// TIA Portal V18 export
FUNCTION "Datalog" : Void   // FC13, LAD
{ S7_Optimized_Access := 'TRUE' }
VERSION : 0.1
// stored: AutoNumber true, IsIECCheckEnabled false, SetENOAutomatically false, UDAEnableTagReadback false
   VAR_TEMP
      "return" : Int;
   END_VAR
   VAR_TEMP   // added for the SCL form of the ladder/FBD networks
      _w1 : Bool;
      _w2 : Bool;
      _w3 : Bool;
      _w4 : Bool;
      _w5 : Bool;
      _w6 : Bool;
      _w7 : Bool;
      _w8 : Bool;
   END_VAR
BEGIN

REGION Network 1
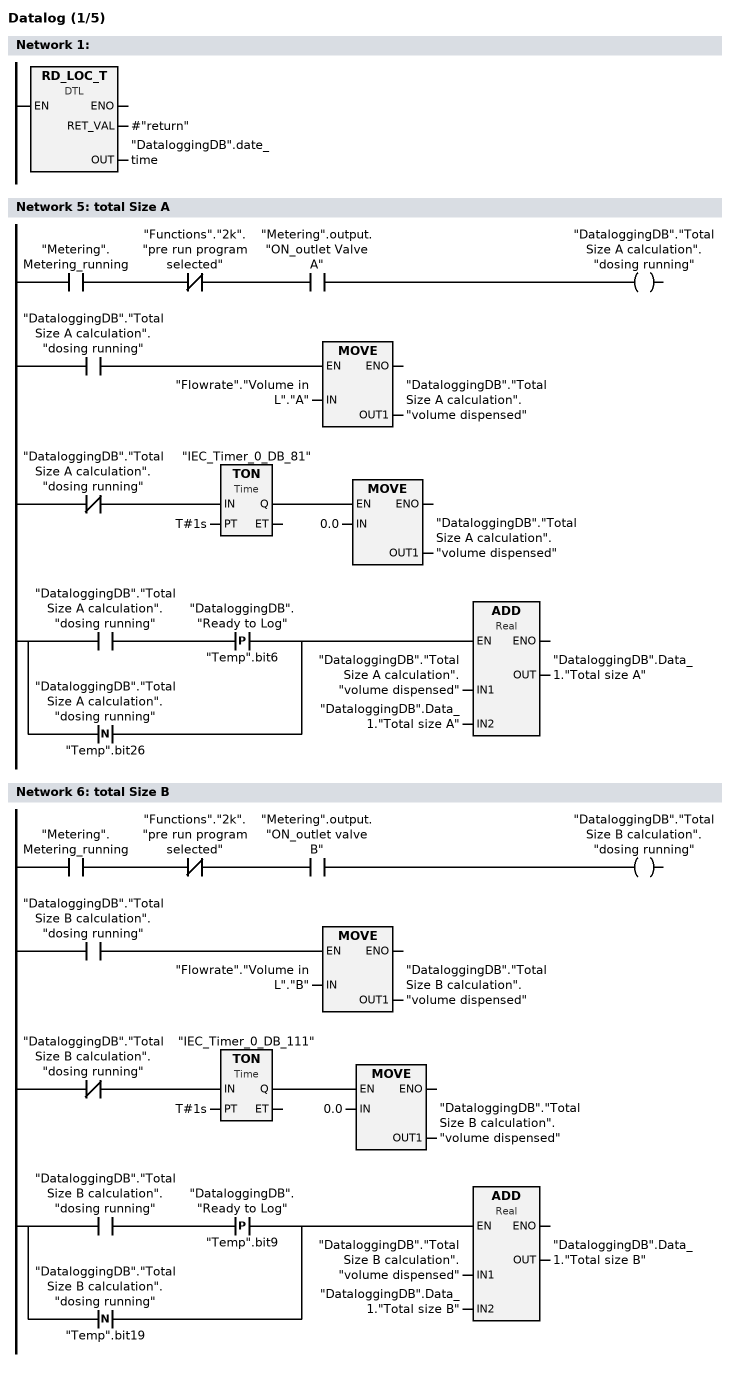
   RUNG wire#powerrail
      { S7_Templates := "date_type := DTL" } RD_LOC_T(RET_VAL => #"return", OUT => "DataloggingDB".date_time)
   END_RUNG
   // the same network as SCL:
   #"return" := RD_LOC_T(OUT => "DataloggingDB".date_time);
END_REGION

REGION Network 2 (SCL)
   IF "DataloggingDB".date_time.DAY <> "DataloggingDB".previous_day THEN
       //"DataloggingDB".day_changed := true;
       "DataloggingDB".totalsizepreviousday:="DataloggingDB".Data_1."Total Size";
       "DataloggingDB".previous_day := "DataloggingDB".date_time.DAY ;
   ELSE
       "DataloggingDB".day_changed := false;
   END_IF;
   IF "DataloggingDB".current_week <> "DataloggingDB".previous_week THEN
       //"DataloggingDB".day_changed := true;
       "DataloggingDB".totalsizepreviousweek := "DataloggingDB".Data_1."Total Size";
       "DataloggingDB".previous_week := "DataloggingDB".current_week;
   ELSE
       "DataloggingDB".day_changed := false;
   END_IF;

   IF "DataloggingDB".date_time.MONTH <> "DataloggingDB".previous_month THEN
       //"DataloggingDB".month_changed := true;
       "DataloggingDB".totalsizepreviousmonth := "DataloggingDB".Data_1."Total Size";
       "DataloggingDB".previous_month := "DataloggingDB".date_time.MONTH;
   ELSE
       "DataloggingDB".month_changed := false;
   END_IF;

   "DataloggingDB".totalsizeday := "DataloggingDB".Data_1."Total Size" - "DataloggingDB".totalsizepreviousday ;
   "DataloggingDB".totalsizeweek := "DataloggingDB".Data_1."Total Size" - "DataloggingDB".totalsizepreviousweek;
   "DataloggingDB".totalsizemonth := "DataloggingDB".Data_1."Total Size" - "DataloggingDB".totalsizepreviousmonth;
END_REGION

REGION Network 3 (SCL): Total Flush A
   IF (("Function Flush"."Control A"."flush running" AND "Functions"."flush selection"."Flush A selected") OR
       "Function Regenaration PGM".Control."metering running" OR
       "Function Ratio check".Control."metering running" OR
       ("Functions"."2k"."pre run program selected" AND "Metering".Metering_running) OR
       "Function Dearing with valve"."Control A"."dearing running") THEN
       "DataloggingDB"."Copy Flush A qty" := true;
   END_IF;

   "R_TRIG_DB_1"(CLK:="DataloggingDB"."Copy Flush A qty" AND NOT ("Function Dearing with valve"."Control A"."dearing running") AND
                 NOT ("Function Regenaration PGM".Control."metering running") AND NOT ("Function Ratio check".Control."metering running") AND
                 NOT ("Functions"."2k"."pre run program selected") AND NOT ("Function Flush"."Control A"."flush running"),
                 Q=>"Temp".bit1);

   IF "R_TRIG_DB_1".Q THEN
       "DataloggingDB".Data_1."Total A flush" := "Flowrate"."Volume in L".mixed +"DataloggingDB".Data_1."Total A flush";
       "DataloggingDB"."Copy Flush A qty" := false;
   END_IF;
END_REGION

REGION Network 4 (SCL)
   IF (("Function Flush"."Control B"."flush running" AND "Functions"."flush selection"."Flush B selected") OR
       "Function Regenaration PGM".Control."metering running" OR
       "Function Ratio check".Control."metering running" OR
       ("Functions"."2k"."pre run program selected" AND "Metering".Metering_running) OR
       "Function Dearing with valve"."Control B"."dearing running") THEN
       "DataloggingDB"."Copy Flush B qty" := true;
   END_IF;

   "R_TRIG_DB_21"(CLK:="DataloggingDB"."Copy Flush B qty" AND NOT ("Function Dearing with valve"."Control B"."dearing running") AND
                  NOT ("Function Regenaration PGM".Control."metering running") AND NOT ("Function Ratio check".Control."metering running") AND
                  NOT ("Functions"."2k"."pre run program selected") AND NOT ("Function Flush"."Control B"."flush running"),
                  Q=>"Temp".bit3);

   IF "R_TRIG_DB_21".Q THEN
       "DataloggingDB".Data_1."Total B flush" := "Flowrate"."Volume in L".mixed + "DataloggingDB".Data_1."Total B flush";
       "DataloggingDB"."Copy Flush B qty" := false;
   END_IF;
END_REGION

REGION Network 5: total Size A
   RUNG wire#powerrail
      Contact( "Metering".Metering_running )
      I_Contact( "Functions"."2k"."pre run program selected" )
      Contact( "Metering".output."ON_outlet Valve A" )
      Coil( "DataloggingDB"."Total Size A calculation"."dosing running" )
   END_RUNG
   RUNG wire#powerrail
      Contact( "DataloggingDB"."Total Size A calculation"."dosing running" )
      Move(in := "Flowrate"."Volume in L"."A", out1 => "DataloggingDB"."Total Size A calculation"."volume dispensed")
   END_RUNG
   RUNG wire#powerrail
      I_Contact( "DataloggingDB"."Total Size A calculation"."dosing running" )
      { S7_Templates := "time_type := Time" } "IEC_Timer_0_DB_81".TON(pt := T#1s, et =>)
      Move(in := 0.0, out1 => "DataloggingDB"."Total Size A calculation"."volume dispensed")
   END_RUNG
   RUNG wire#powerrail
      Contact( "DataloggingDB"."Total Size A calculation"."dosing running" )
      P_Contact(operand := "DataloggingDB"."Ready to Log", bit := "Temp".bit6)
      wire#w1
      { S7_Templates := "SrcType := Real" } Add(in1 := "DataloggingDB"."Total Size A calculation"."volume dispensed", in2 := "DataloggingDB".Data_1."Total size A", out => "DataloggingDB".Data_1."Total size A")
   END_RUNG
   RUNG wire#powerrail
      N_Contact(operand := "DataloggingDB"."Total Size A calculation"."dosing running", bit := "Temp".bit26)
   END_RUNG wire#w1
   // the same network as SCL:
   "DataloggingDB"."Total Size A calculation"."dosing running" := "Metering".Metering_running AND NOT "Functions"."2k"."pre run program selected" AND "Metering".output."ON_outlet Valve A";
   IF "DataloggingDB"."Total Size A calculation"."dosing running" THEN
       "DataloggingDB"."Total Size A calculation"."volume dispensed" := "Flowrate"."Volume in L"."A";
   END_IF;
   "IEC_Timer_0_DB_81".TON(IN := NOT "DataloggingDB"."Total Size A calculation"."dosing running", PT := T#1s);
   IF "IEC_Timer_0_DB_81".Q THEN
       "DataloggingDB"."Total Size A calculation"."volume dispensed" := 0.0;
   END_IF;
   #_w1 := "DataloggingDB"."Total Size A calculation"."dosing running" AND "DataloggingDB"."Ready to Log" AND NOT "Temp".bit6;   // rising edge of "DataloggingDB"."Ready to Log"
   "Temp".bit6 := "DataloggingDB"."Ready to Log";
   #_w2 := NOT "DataloggingDB"."Total Size A calculation"."dosing running" AND "Temp".bit26;   // falling edge of "DataloggingDB"."Total Size A calculation"."dosing running"
   "Temp".bit26 := "DataloggingDB"."Total Size A calculation"."dosing running";
   IF #_w1 OR #_w2 THEN
       "DataloggingDB".Data_1."Total size A" := "DataloggingDB"."Total Size A calculation"."volume dispensed" + "DataloggingDB".Data_1."Total size A";
   END_IF;
END_REGION

REGION Network 6: total Size B
   RUNG wire#powerrail
      Contact( "Metering".Metering_running )
      I_Contact( "Functions"."2k"."pre run program selected" )
      Contact( "Metering".output."ON_outlet valve B" )
      Coil( "DataloggingDB"."Total Size B calculation"."dosing running" )
   END_RUNG
   RUNG wire#powerrail
      Contact( "DataloggingDB"."Total Size B calculation"."dosing running" )
      Move(in := "Flowrate"."Volume in L"."B", out1 => "DataloggingDB"."Total Size B calculation"."volume dispensed")
   END_RUNG
   RUNG wire#powerrail
      I_Contact( "DataloggingDB"."Total Size B calculation"."dosing running" )
      { S7_Templates := "time_type := Time" } "IEC_Timer_0_DB_111".TON(pt := T#1s, et =>)
      Move(in := 0.0, out1 => "DataloggingDB"."Total Size B calculation"."volume dispensed")
   END_RUNG
   RUNG wire#powerrail
      Contact( "DataloggingDB"."Total Size B calculation"."dosing running" )
      P_Contact(operand := "DataloggingDB"."Ready to Log", bit := "Temp".bit9)
      wire#w1
      { S7_Templates := "SrcType := Real" } Add(in1 := "DataloggingDB"."Total Size B calculation"."volume dispensed", in2 := "DataloggingDB".Data_1."Total size B", out => "DataloggingDB".Data_1."Total size B")
   END_RUNG
   RUNG wire#powerrail
      N_Contact(operand := "DataloggingDB"."Total Size B calculation"."dosing running", bit := "Temp".bit19)
   END_RUNG wire#w1
   // the same network as SCL:
   "DataloggingDB"."Total Size B calculation"."dosing running" := "Metering".Metering_running AND NOT "Functions"."2k"."pre run program selected" AND "Metering".output."ON_outlet valve B";
   IF "DataloggingDB"."Total Size B calculation"."dosing running" THEN
       "DataloggingDB"."Total Size B calculation"."volume dispensed" := "Flowrate"."Volume in L"."B";
   END_IF;
   "IEC_Timer_0_DB_111".TON(IN := NOT "DataloggingDB"."Total Size B calculation"."dosing running", PT := T#1s);
   IF "IEC_Timer_0_DB_111".Q THEN
       "DataloggingDB"."Total Size B calculation"."volume dispensed" := 0.0;
   END_IF;
   #_w1 := "DataloggingDB"."Total Size B calculation"."dosing running" AND "DataloggingDB"."Ready to Log" AND NOT "Temp".bit9;   // rising edge of "DataloggingDB"."Ready to Log"
   "Temp".bit9 := "DataloggingDB"."Ready to Log";
   #_w2 := NOT "DataloggingDB"."Total Size B calculation"."dosing running" AND "Temp".bit19;   // falling edge of "DataloggingDB"."Total Size B calculation"."dosing running"
   "Temp".bit19 := "DataloggingDB"."Total Size B calculation"."dosing running";
   IF #_w1 OR #_w2 THEN
       "DataloggingDB".Data_1."Total size B" := "DataloggingDB"."Total Size B calculation"."volume dispensed" + "DataloggingDB".Data_1."Total size B";
   END_IF;
END_REGION

REGION Network 7: Total size
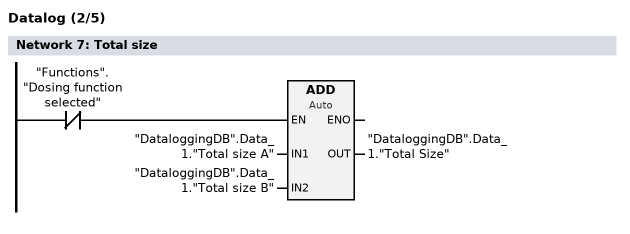
   RUNG wire#powerrail
      I_Contact( "Functions"."Dosing function selected" )
      Add(in1 := "DataloggingDB".Data_1."Total size A", in2 := "DataloggingDB".Data_1."Total size B", out => "DataloggingDB".Data_1."Total Size")
   END_RUNG
   // the same network as SCL:
   IF NOT "Functions"."Dosing function selected" THEN
       "DataloggingDB".Data_1."Total Size" := "DataloggingDB".Data_1."Total size A" + "DataloggingDB".Data_1."Total size B";
   END_IF;
END_REGION

REGION Network 8: Metering Size
END_REGION

REGION Network 9: Shot Size A
END_REGION

REGION Network 10: Shot Size B
END_REGION

REGION Network 11: Mixing Ratio
END_REGION

REGION Network 12: ratio Min
END_REGION

REGION Network 13: ratio Max
END_REGION

REGION Network 14: Volume_Dispensed
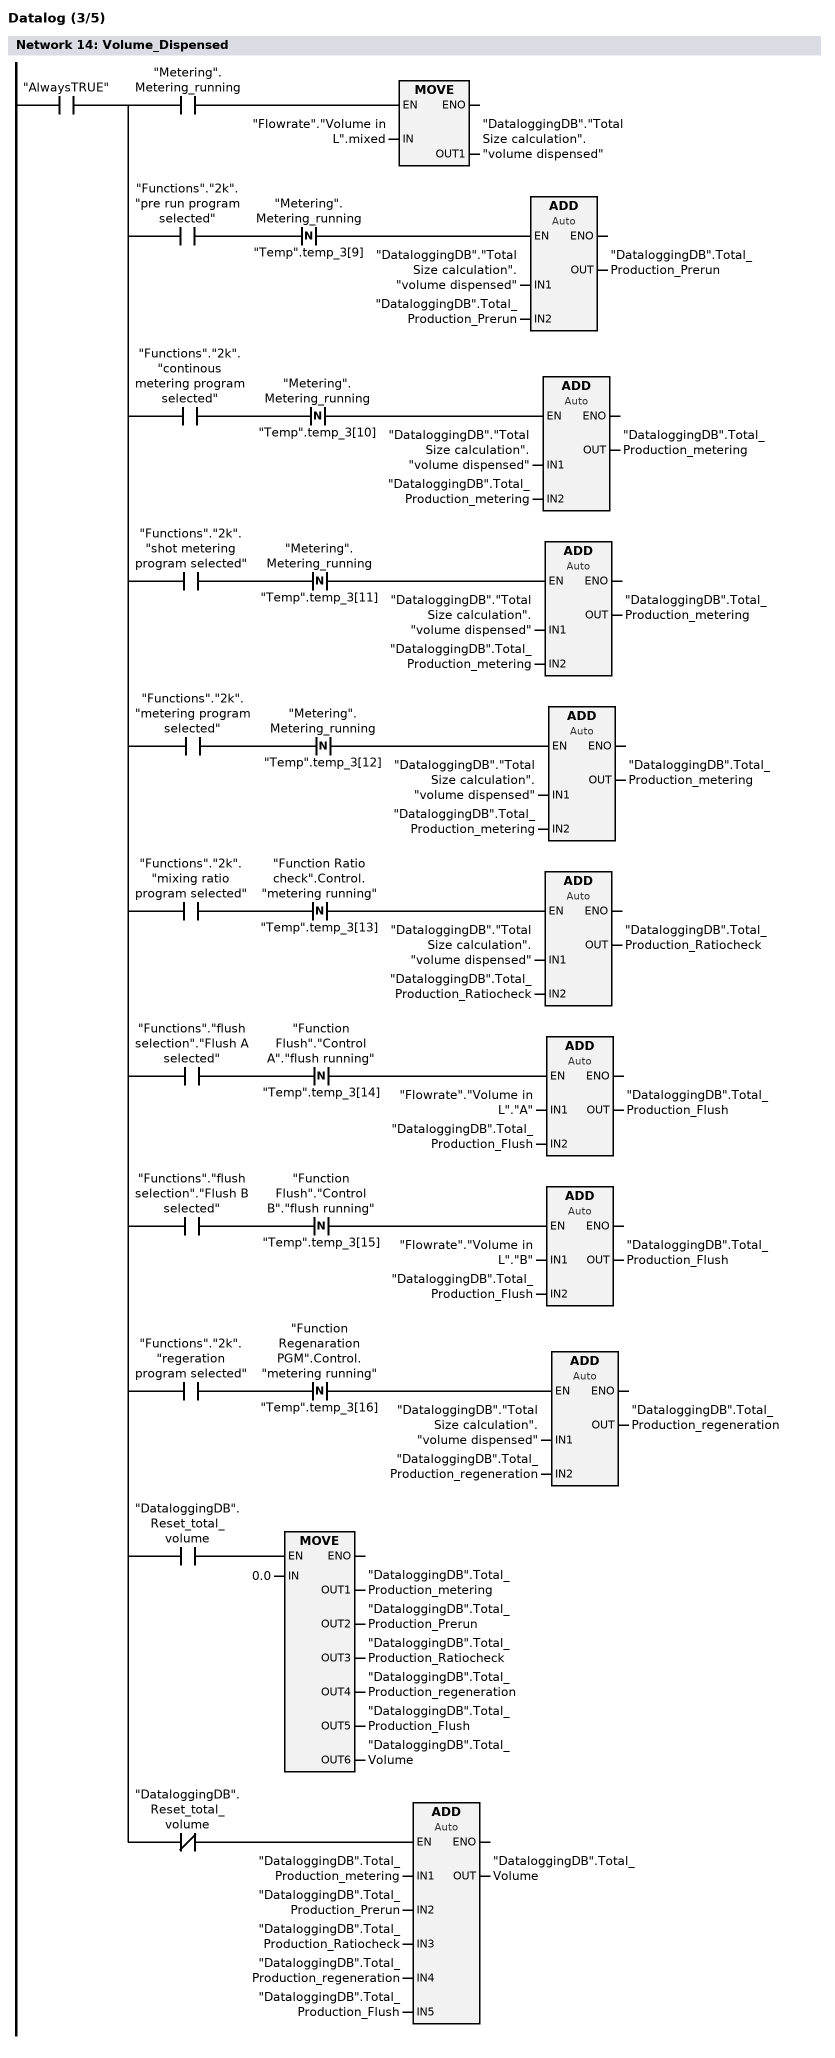
   RUNG wire#powerrail
      Contact( "AlwaysTRUE" )
      wire#w1
      Contact( "Metering".Metering_running )
      Move(in := "Flowrate"."Volume in L".mixed, out1 => "DataloggingDB"."Total Size calculation"."volume dispensed")
   END_RUNG
   RUNG wire#w1
      Contact( "Functions"."2k"."pre run program selected" )
      N_Contact(operand := "Metering".Metering_running, bit := "Temp".temp_3[9])
      Add(in1 := "DataloggingDB"."Total Size calculation"."volume dispensed", in2 := "DataloggingDB".Total_Production_Prerun, out => "DataloggingDB".Total_Production_Prerun)
   END_RUNG
   RUNG wire#w1
      Contact( "Functions"."2k"."continous metering program selected" )
      N_Contact(operand := "Metering".Metering_running, bit := "Temp".temp_3[10])
      Add(in1 := "DataloggingDB"."Total Size calculation"."volume dispensed", in2 := "DataloggingDB".Total_Production_metering, out => "DataloggingDB".Total_Production_metering)
   END_RUNG
   RUNG wire#w1
      Contact( "Functions"."2k"."shot metering program selected" )
      N_Contact(operand := "Metering".Metering_running, bit := "Temp".temp_3[11])
      Add(in1 := "DataloggingDB"."Total Size calculation"."volume dispensed", in2 := "DataloggingDB".Total_Production_metering, out => "DataloggingDB".Total_Production_metering)
   END_RUNG
   RUNG wire#w1
      Contact( "Functions"."2k"."metering program selected" )
      N_Contact(operand := "Metering".Metering_running, bit := "Temp".temp_3[12])
      Add(in1 := "DataloggingDB"."Total Size calculation"."volume dispensed", in2 := "DataloggingDB".Total_Production_metering, out => "DataloggingDB".Total_Production_metering)
   END_RUNG
   RUNG wire#w1
      Contact( "Functions"."2k"."mixing ratio program selected" )
      N_Contact(operand := "Function Ratio check".Control."metering running", bit := "Temp".temp_3[13])
      Add(in1 := "DataloggingDB"."Total Size calculation"."volume dispensed", in2 := "DataloggingDB".Total_Production_Ratiocheck, out => "DataloggingDB".Total_Production_Ratiocheck)
   END_RUNG
   RUNG wire#w1
      Contact( "Functions"."flush selection"."Flush A selected" )
      N_Contact(operand := "Function Flush"."Control A"."flush running", bit := "Temp".temp_3[14])
      Add(in1 := "Flowrate"."Volume in L"."A", in2 := "DataloggingDB".Total_Production_Flush, out => "DataloggingDB".Total_Production_Flush)
   END_RUNG
   RUNG wire#w1
      Contact( "Functions"."flush selection"."Flush B selected" )
      N_Contact(operand := "Function Flush"."Control B"."flush running", bit := "Temp".temp_3[15])
      Add(in1 := "Flowrate"."Volume in L"."B", in2 := "DataloggingDB".Total_Production_Flush, out => "DataloggingDB".Total_Production_Flush)
   END_RUNG
   RUNG wire#w1
      Contact( "Functions"."2k"."regeration program selected" )
      N_Contact(operand := "Function Regenaration PGM".Control."metering running", bit := "Temp".temp_3[16])
      Add(in1 := "DataloggingDB"."Total Size calculation"."volume dispensed", in2 := "DataloggingDB".Total_Production_regeneration, out => "DataloggingDB".Total_Production_regeneration)
   END_RUNG
   RUNG wire#w1
      Contact( "DataloggingDB".Reset_total_volume )
      Move(in := 0.0, out1 => "DataloggingDB".Total_Production_metering, out2 => "DataloggingDB".Total_Production_Prerun, out3 => "DataloggingDB".Total_Production_Ratiocheck, out4 => "DataloggingDB".Total_Production_regeneration, out5 => "DataloggingDB".Total_Production_Flush, out6 => "DataloggingDB".Total_Volume)
   END_RUNG
   RUNG wire#w1
      I_Contact( "DataloggingDB".Reset_total_volume )
      Add(in1 := "DataloggingDB".Total_Production_metering, in2 := "DataloggingDB".Total_Production_Prerun, in3 := "DataloggingDB".Total_Production_Ratiocheck, in4 := "DataloggingDB".Total_Production_regeneration, in5 := "DataloggingDB".Total_Production_Flush, out => "DataloggingDB".Total_Volume)
   END_RUNG
   // the same network as SCL:
   IF "AlwaysTRUE" AND "Metering".Metering_running THEN
       "DataloggingDB"."Total Size calculation"."volume dispensed" := "Flowrate"."Volume in L".mixed;
   END_IF;
   #_w1 := "AlwaysTRUE" AND "Functions"."2k"."pre run program selected" AND NOT "Metering".Metering_running AND "Temp".temp_3[9];   // falling edge of "Metering".Metering_running
   "Temp".temp_3[9] := "Metering".Metering_running;
   IF #_w1 THEN
       "DataloggingDB".Total_Production_Prerun := "DataloggingDB"."Total Size calculation"."volume dispensed" + "DataloggingDB".Total_Production_Prerun;
   END_IF;
   #_w2 := "AlwaysTRUE" AND "Functions"."2k"."continous metering program selected" AND NOT "Metering".Metering_running AND "Temp".temp_3[10];   // falling edge of "Metering".Metering_running
   "Temp".temp_3[10] := "Metering".Metering_running;
   IF #_w2 THEN
       "DataloggingDB".Total_Production_metering := "DataloggingDB"."Total Size calculation"."volume dispensed" + "DataloggingDB".Total_Production_metering;
   END_IF;
   #_w3 := "AlwaysTRUE" AND "Functions"."2k"."shot metering program selected" AND NOT "Metering".Metering_running AND "Temp".temp_3[11];   // falling edge of "Metering".Metering_running
   "Temp".temp_3[11] := "Metering".Metering_running;
   IF #_w3 THEN
       "DataloggingDB".Total_Production_metering := "DataloggingDB"."Total Size calculation"."volume dispensed" + "DataloggingDB".Total_Production_metering;
   END_IF;
   #_w4 := "AlwaysTRUE" AND "Functions"."2k"."metering program selected" AND NOT "Metering".Metering_running AND "Temp".temp_3[12];   // falling edge of "Metering".Metering_running
   "Temp".temp_3[12] := "Metering".Metering_running;
   IF #_w4 THEN
       "DataloggingDB".Total_Production_metering := "DataloggingDB"."Total Size calculation"."volume dispensed" + "DataloggingDB".Total_Production_metering;
   END_IF;
   #_w5 := "AlwaysTRUE" AND "Functions"."2k"."mixing ratio program selected" AND NOT "Function Ratio check".Control."metering running" AND "Temp".temp_3[13];   // falling edge of "Function Ratio check".Control."metering running"
   "Temp".temp_3[13] := "Function Ratio check".Control."metering running";
   IF #_w5 THEN
       "DataloggingDB".Total_Production_Ratiocheck := "DataloggingDB"."Total Size calculation"."volume dispensed" + "DataloggingDB".Total_Production_Ratiocheck;
   END_IF;
   #_w6 := "AlwaysTRUE" AND "Functions"."flush selection"."Flush A selected" AND NOT "Function Flush"."Control A"."flush running" AND "Temp".temp_3[14];   // falling edge of "Function Flush"."Control A"."flush running"
   "Temp".temp_3[14] := "Function Flush"."Control A"."flush running";
   IF #_w6 THEN
       "DataloggingDB".Total_Production_Flush := "Flowrate"."Volume in L"."A" + "DataloggingDB".Total_Production_Flush;
   END_IF;
   #_w7 := "AlwaysTRUE" AND "Functions"."flush selection"."Flush B selected" AND NOT "Function Flush"."Control B"."flush running" AND "Temp".temp_3[15];   // falling edge of "Function Flush"."Control B"."flush running"
   "Temp".temp_3[15] := "Function Flush"."Control B"."flush running";
   IF #_w7 THEN
       "DataloggingDB".Total_Production_Flush := "Flowrate"."Volume in L"."B" + "DataloggingDB".Total_Production_Flush;
   END_IF;
   #_w8 := "AlwaysTRUE" AND "Functions"."2k"."regeration program selected" AND NOT "Function Regenaration PGM".Control."metering running" AND "Temp".temp_3[16];   // falling edge of "Function Regenaration PGM".Control."metering running"
   "Temp".temp_3[16] := "Function Regenaration PGM".Control."metering running";
   IF #_w8 THEN
       "DataloggingDB".Total_Production_regeneration := "DataloggingDB"."Total Size calculation"."volume dispensed" + "DataloggingDB".Total_Production_regeneration;
   END_IF;
   IF "AlwaysTRUE" AND "DataloggingDB".Reset_total_volume THEN
       "DataloggingDB".Total_Production_metering := 0.0;
       "DataloggingDB".Total_Production_Prerun := 0.0;
       "DataloggingDB".Total_Production_Ratiocheck := 0.0;
       "DataloggingDB".Total_Production_regeneration := 0.0;
       "DataloggingDB".Total_Production_Flush := 0.0;
       "DataloggingDB".Total_Volume := 0.0;
   END_IF;
   IF "AlwaysTRUE" AND NOT "DataloggingDB".Reset_total_volume THEN
       "DataloggingDB".Total_Volume := "DataloggingDB".Total_Production_metering + "DataloggingDB".Total_Production_Prerun + "DataloggingDB".Total_Production_Ratiocheck + "DataloggingDB".Total_Production_regeneration + "DataloggingDB".Total_Production_Flush;
   END_IF;
END_REGION

REGION Network 15 (SCL)
   IF NOT ("Functions"."Dosing Running") THEN
       "event For datalogging"."event number" := 1; //Event machine idle
   ELSIF "Functions"."2k"."metering program selected" AND "Metering".Metering_running THEN
       "event For datalogging"."event number" := 2; //Event metering program running
   ELSIF "Function Ratio check".Control."metering running" THEN
       "event For datalogging"."event number" := 3; //Event Ratio check program running
   ELSIF "Functions"."2k"."shot metering program selected" AND "Metering".Metering_running THEN
       "event For datalogging"."event number" := 4; //Event metering shot running
   ELSIF "Functions"."2k"."continous metering program selected" AND "Metering".Metering_running THEN
       "event For datalogging"."event number" := 5; //Event metering Continuous metering running
   ELSIF "Functions"."2k"."pre run program selected" AND "Metering".Metering_running THEN
       "event For datalogging"."event number" := 6; //Event "Metering" Pre run running
   ELSIF "Function Flush"."Control A"."flush running" THEN
       "event For datalogging"."event number" := 7; // Event metering Flush running
   ELSIF "Function Dearing with valve"."Control A"."dearing running" OR "Function Dearing with valve"."Control B"."dearing running" THEN
       "event For datalogging"."event number" := 8; // Event deaerate running
   ELSIF "Faults&warnings"."Critical Alarm metering A&B" THEN
       "event For datalogging"."event number" := 9; // Event Machine fault
   ELSIF "Function Regenaration PGM".Control."metering running" THEN
       "event For datalogging"."event number" := 11; // Event regeneration running
   ELSIF "metering Completed" THEN
       "event For datalogging"."event number" := 12; // dosing completed
   END_IF;

   "DataloggingDB".Data.Function := "event For datalogging".Function_String["event For datalogging"."event number"];
END_REGION

REGION Network 16: Function
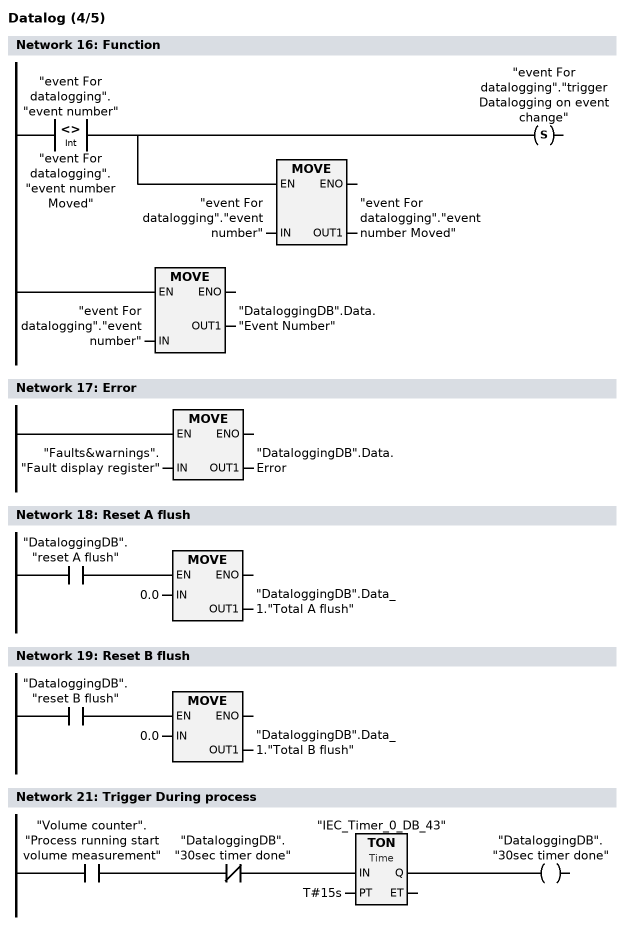
   RUNG wire#powerrail
      { S7_Templates := "SrcType := Int" } NE_Contact(in1 := "event For datalogging"."event number", in2 := "event For datalogging"."event number Moved")
      wire#w1
      S_Coil( "event For datalogging"."trigger Datalogging on event change" )
   END_RUNG
   RUNG wire#w1
      Move(in := "event For datalogging"."event number", out1 => "event For datalogging"."event number Moved")
   END_RUNG
   RUNG wire#powerrail
      Move(in := "event For datalogging"."event number", out1 => "DataloggingDB".Data."Event Number")
   END_RUNG
   // the same network as SCL:
   IF "event For datalogging"."event number" <> "event For datalogging"."event number Moved" THEN
       "event For datalogging"."trigger Datalogging on event change" := TRUE;
       "event For datalogging"."event number Moved" := "event For datalogging"."event number";
   END_IF;
   "DataloggingDB".Data."Event Number" := "event For datalogging"."event number";
END_REGION

REGION Network 17: Error
   RUNG wire#powerrail
      Move(in := "Faults&warnings"."Fault display register", out1 => "DataloggingDB".Data.Error)
   END_RUNG
   // the same network as SCL:
   "DataloggingDB".Data.Error := "Faults&warnings"."Fault display register";
END_REGION

REGION Network 18: Reset A flush
   RUNG wire#powerrail
      Contact( "DataloggingDB"."reset A flush" )
      Move(in := 0.0, out1 => "DataloggingDB".Data_1."Total A flush")
   END_RUNG
   // the same network as SCL:
   IF "DataloggingDB"."reset A flush" THEN "DataloggingDB".Data_1."Total A flush" := 0.0; END_IF;
END_REGION

REGION Network 19: Reset B flush
   RUNG wire#powerrail
      Contact( "DataloggingDB"."reset B flush" )
      Move(in := 0.0, out1 => "DataloggingDB".Data_1."Total B flush")
   END_RUNG
   // the same network as SCL:
   IF "DataloggingDB"."reset B flush" THEN "DataloggingDB".Data_1."Total B flush" := 0.0; END_IF;
END_REGION

REGION Network 20 (SCL): Reset total size
   IF "DataloggingDB"."reset total Size" THEN
       "DataloggingDB".Data_1."Total size A" := 0;
       "DataloggingDB".Data_1."Total size B" := 0;
       "DataloggingDB".totalsizeday := 0;
       "DataloggingDB".totalsizepreviousday := 0;
       "DataloggingDB".totalsizeweek := 0;
       "DataloggingDB".totalsizepreviousweek := 0;
       "DataloggingDB".totalsizemonth := 0;
       "DataloggingDB".totalsizepreviousmonth := 0;
       "DataloggingDB"."reset total Size" := FALSE;
   END_IF;
END_REGION

REGION Network 21: Trigger During process
   RUNG wire#powerrail
      Contact( "Volume counter"."Process running start volume measurement" )
      I_Contact( "DataloggingDB"."30sec timer done" )
      { S7_Templates := "time_type := Time" } "IEC_Timer_0_DB_43".TON(pt := T#15s, et =>)
      Coil( "DataloggingDB"."30sec timer done" )
   END_RUNG
   // the same network as SCL:
   "IEC_Timer_0_DB_43".TON(IN := "Volume counter"."Process running start volume measurement" AND NOT "DataloggingDB"."30sec timer done",
                           PT := T#15s);
   "DataloggingDB"."30sec timer done" := "IEC_Timer_0_DB_43".Q;
END_REGION

REGION Network 22: trigger data logging
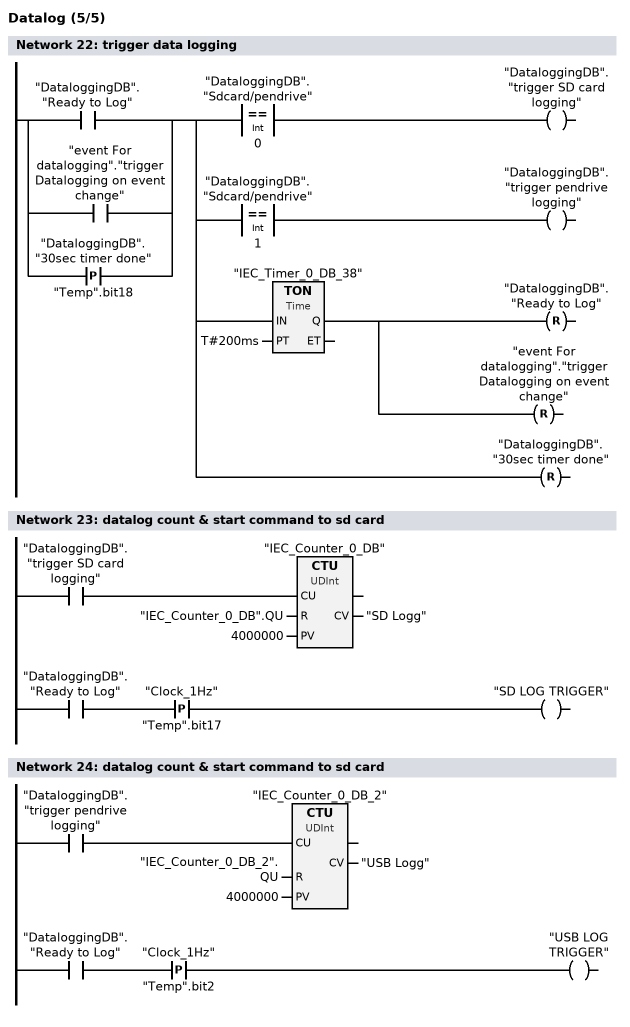
   RUNG wire#powerrail
      Contact( "DataloggingDB"."Ready to Log" )
      wire#w1
      { S7_Templates := "SrcType := Int" } EQ_Contact(in1 := "DataloggingDB"."Sdcard/pendrive", in2 := 0)
      Coil( "DataloggingDB"."trigger SD card logging" )
   END_RUNG
   RUNG wire#powerrail
      Contact( "event For datalogging"."trigger Datalogging on event change" )
   END_RUNG wire#w1
   RUNG wire#powerrail
      P_Contact(operand := "DataloggingDB"."30sec timer done", bit := "Temp".bit18)
   END_RUNG wire#w1
   RUNG wire#w1
      { S7_Templates := "SrcType := Int" } EQ_Contact(in1 := "DataloggingDB"."Sdcard/pendrive", in2 := 1)
      Coil( "DataloggingDB"."trigger pendrive logging" )
   END_RUNG
   RUNG wire#w1
      { S7_Templates := "time_type := Time" } "IEC_Timer_0_DB_38".TON(pt := T#200ms, et =>)
      wire#w2
      R_Coil( "DataloggingDB"."Ready to Log" )
   END_RUNG
   RUNG wire#w2
      R_Coil( "event For datalogging"."trigger Datalogging on event change" )
   END_RUNG
   RUNG wire#w1
      R_Coil( "DataloggingDB"."30sec timer done" )
   END_RUNG
   // the same network as SCL:
   #_w1 := "DataloggingDB"."30sec timer done" AND NOT "Temp".bit18;   // rising edge of "DataloggingDB"."30sec timer done"
   "Temp".bit18 := "DataloggingDB"."30sec timer done";
   #_w2 := "DataloggingDB"."Ready to Log" OR "event For datalogging"."trigger Datalogging on event change" OR #_w1;
   "DataloggingDB"."trigger SD card logging" := #_w2 AND ("DataloggingDB"."Sdcard/pendrive" = 0);
   "DataloggingDB"."trigger pendrive logging" := #_w2 AND ("DataloggingDB"."Sdcard/pendrive" = 1);
   "IEC_Timer_0_DB_38".TON(IN := #_w2, PT := T#200ms);
   IF "IEC_Timer_0_DB_38".Q THEN
       "DataloggingDB"."Ready to Log" := FALSE;
       "event For datalogging"."trigger Datalogging on event change" := FALSE;
   END_IF;
   IF #_w2 THEN "DataloggingDB"."30sec timer done" := FALSE; END_IF;
END_REGION

REGION Network 23: datalog count & start command to sd card
   RUNG wire#powerrail
      Contact( "DataloggingDB"."trigger SD card logging" )
      { S7_Templates := "value_type := UDInt" } "IEC_Counter_0_DB".CTU(r := "IEC_Counter_0_DB".QU, pv := 4000000, cv => "SD Logg")
   END_RUNG
   RUNG wire#powerrail
      Contact( "DataloggingDB"."Ready to Log" )
      P_Contact(operand := "Clock_1Hz", bit := "Temp".bit17)
      Coil( "SD LOG TRIGGER" )
   END_RUNG
   // the same network as SCL:
   "IEC_Counter_0_DB".CTU(CU := "DataloggingDB"."trigger SD card logging",
                          R := "IEC_Counter_0_DB".QU,
                          PV := 4000000,
                          CV => "SD Logg");
   #_w1 := "DataloggingDB"."Ready to Log" AND "Clock_1Hz" AND NOT "Temp".bit17;   // rising edge of "Clock_1Hz"
   "Temp".bit17 := "Clock_1Hz";
   "SD LOG TRIGGER" := #_w1;
END_REGION

REGION Network 24: datalog count & start command to sd card
   RUNG wire#powerrail
      Contact( "DataloggingDB"."trigger pendrive logging" )
      { S7_Templates := "value_type := UDInt" } "IEC_Counter_0_DB_2".CTU(r := "IEC_Counter_0_DB_2".QU, pv := 4000000, cv => "USB Logg")
   END_RUNG
   RUNG wire#powerrail
      Contact( "DataloggingDB"."Ready to Log" )
      P_Contact(operand := "Clock_1Hz", bit := "Temp".bit2)
      Coil( "USB LOG TRIGGER" )
   END_RUNG
   // the same network as SCL:
   "IEC_Counter_0_DB_2".CTU(CU := "DataloggingDB"."trigger pendrive logging",
                           R := "IEC_Counter_0_DB_2".QU,
                           PV := 4000000,
                           CV => "USB Logg");
   #_w1 := "DataloggingDB"."Ready to Log" AND "Clock_1Hz" AND NOT "Temp".bit2;   // rising edge of "Clock_1Hz"
   "Temp".bit2 := "Clock_1Hz";
   "USB LOG TRIGGER" := #_w1;
END_REGION
END_FUNCTION
